(* Logix 5000 project; controller p65 vendor 1 type 14 code 85 rev 20.11; software revision 20.01; part 5 of 7 *)
(* tags used below, declared in another part *)
   DCMicroGridisInOperation : ALIAS FOR DINT00_23.8;
   DCMicroGridisSimulating : ALIAS FOR DINT00_23.10;
   House05accountBalance : ALIAS FOR REAL00_167;
   House05accountDepositRate : ALIAS FOR REAL00_168;
   House05Bclose : ALIAS FOR Local:3:O.Data.4;
   House05BcloseHILS : ALIAS FOR plc1_local_6[0].4;
   House05BcloseProxy : ALIAS FOR DINT00_31.1;
   House05BintReqClose : ALIAS FOR DINT00_31.2;
   House05BisClosed : ALIAS FOR DINT00_31.3;
   House05BisOpen : ALIAS FOR DINT00_31.4;
   House05BreqClose : ALIAS FOR DINT00_31.5;
   House05BreqOpen : ALIAS FOR DINT00_31.6;
   House05commandChanged : ALIAS FOR DINT00_31.7;
   House05commandChangedTimer : ALIAS FOR CLTIMER00_78;
   House05current : ALIAS FOR REAL00_169;
   House05currentHILS : ALIAS FOR plc1_local_2[4];
   House05currentRaw : ALIAS FOR Local:2:I.Ch0Data;
   House05deadband : ALIAS FOR REAL00_170;
   House05depositTimer : ALIAS FOR CLTIMER00_79;
   House05DisconnectPowerEventFail : ALIAS FOR DINT00_31.8;
   House05DisconnectPowerEventSuccess : ALIAS FOR DINT00_31.9;
   House05DisconnectPowerFailTimer : ALIAS FOR CLTIMER00_80;
   House05DisconnectPowerInProcess : ALIAS FOR DINT00_31.10;
   House05DisconnectPowerMsg : ALIAS FOR MESSAGE00_20;
   House05DisconnectPowerSuccessTimer : ALIAS FOR CLTIMER00_81;
   House05failedToConnect : ALIAS FOR DINT00_31.11;
   House05failedToDisconnect : ALIAS FOR DINT00_31.12;
   House05fundsAvailable : ALIAS FOR DINT00_31.13;
   House05incrementToAdd : ALIAS FOR REAL00_171;
   House05incrementToSubtract : ALIAS FOR REAL00_172;
   House05intReqConnect : ALIAS FOR DINT00_31.14;
   House05isConnected : ALIAS FOR DINT00_31.15;
   House05isDisconnected : ALIAS FOR DINT00_31.16;
   House05minBalance : ALIAS FOR REAL00_174;
   House05minBalanceToReconnect : ALIAS FOR REAL00_175;
   House05minTime : ALIAS FOR REAL00_176;
   House05powerRate : ALIAS FOR REAL00_177;
   House05powerRateMax : REAL;
   House05PurchasePowerEventFail : ALIAS FOR DINT00_31.17;
   House05PurchasePowerEventSuccess : ALIAS FOR DINT00_31.18;
   House05PurchasePowerFailTimer : ALIAS FOR CLTIMER00_82;
   House05PurchasePowerInProcess : ALIAS FOR DINT00_31.19;
   House05PurchasePowerMsg : ALIAS FOR MESSAGE00_21;
   House05PurchasePowerSuccessTimer : ALIAS FOR CLTIMER00_83;
   House05reqConnect : ALIAS FOR DINT00_31.20;
   House05reqDisconnect : ALIAS FOR DINT00_31.21;
   House05runningOut : ALIAS FOR DINT00_31.22;
   House05spendingRate : ALIAS FOR REAL00_178;
   House05timeRemaining : ALIAS FOR REAL00_179;
   House05usageTimer : ALIAS FOR CLTIMER00_84;
   Load01accountBalance : ALIAS FOR REAL00_37;
   Load01accountDepositRate : ALIAS FOR REAL00_38;
   Load01Bclose : ALIAS FOR Local:3:O.Data.5;
   Load01BcloseHILS : ALIAS FOR plc1_local_6[0].5;
   Load01BcloseProxy : ALIAS FOR DINT00_23.31;
   Load01BintReqClose : ALIAS FOR DINT00_24.0;
   Load01BisClosed : ALIAS FOR DINT00_24.1;
   Load01BisOpen : ALIAS FOR DINT00_24.2;
   Load01BreqClose : ALIAS FOR DINT00_24.3;
   Load01BreqOpen : ALIAS FOR DINT00_24.4;
   Load01commandChanged : ALIAS FOR DINT00_24.5;
   Load01commandChangedTimer : ALIAS FOR CLTIMER00_9;
   Load01current : ALIAS FOR REAL00_39;
   Load01currentHILS : ALIAS FOR plc1_local_2[5];
   Load01currentRaw : ALIAS FOR Local:2:I.Ch2Data;
   Load01deadband : ALIAS FOR REAL00_40;
   Load01depositTimer : ALIAS FOR CLTIMER00_10;
   Load01DisconnectPowerEventFail : ALIAS FOR DINT00_24.6;
   Load01DisconnectPowerEventSuccess : ALIAS FOR DINT00_24.7;
   Load01DisconnectPowerFailTimer : ALIAS FOR CLTIMER00_11;
   Load01DisconnectPowerInProcess : ALIAS FOR DINT00_24.8;
   Load01DisconnectPowerMsg : ALIAS FOR MESSAGE00_1;
   Load01DisconnectPowerSuccessTimer : ALIAS FOR CLTIMER00_12;
   Load01failedToConnect : ALIAS FOR DINT00_24.9;
   Load01failedToDisconnect : ALIAS FOR DINT00_24.10;
   Load01fundsAvailable : ALIAS FOR DINT00_24.11;
   Load01incrementToAdd : ALIAS FOR REAL00_41;
   Load01incrementToSubtract : ALIAS FOR REAL00_42;
   Load01intReqConnect : ALIAS FOR DINT00_24.12;
   Load01isConnected : ALIAS FOR DINT00_24.13;
   Load01isDisconnected : ALIAS FOR DINT00_24.14;
   Load01minBalance : ALIAS FOR REAL00_44;
   Load01minBalanceToReconnect : ALIAS FOR REAL00_45;
   Load01minTime : ALIAS FOR REAL00_46;
   Load01powerRate : ALIAS FOR REAL00_47;
   Load01powerRateMax : REAL;
   Load01PurchasePowerEventFail : ALIAS FOR DINT00_24.15;
   Load01PurchasePowerEventSuccess : ALIAS FOR DINT00_24.16;
   Load01PurchasePowerFailTimer : ALIAS FOR CLTIMER00_13;
   Load01PurchasePowerInProcess : ALIAS FOR DINT00_24.17;
   Load01PurchasePowerMsg : ALIAS FOR MESSAGE00_2;
   Load01PurchasePowerSuccessTimer : ALIAS FOR CLTIMER00_14;
   Load01reqConnect : ALIAS FOR DINT00_24.18;
   Load01reqDisconnect : ALIAS FOR DINT00_24.19;
   Load01runningOut : ALIAS FOR DINT00_24.20;
   Load01spendingRate : ALIAS FOR REAL00_48;
   Load01timeRemaining : ALIAS FOR REAL00_49;
   Load01usageTimer : ALIAS FOR CLTIMER00_15;
   Load02accountBalance : ALIAS FOR REAL00_50;
   Load02accountDepositRate : ALIAS FOR REAL00_51;
   Load02Bclose : ALIAS FOR Local:3:O.Data.6;
   Load02BcloseHILS : ALIAS FOR plc1_local_6[0].6;
   Load02BcloseProxy : ALIAS FOR DINT00_24.21;
   Load02BintReqClose : ALIAS FOR DINT00_24.22;
   Load02BisClosed : ALIAS FOR DINT00_24.23;
   Load02BisOpen : ALIAS FOR DINT00_24.24;
   Load02BreqClose : ALIAS FOR DINT00_24.25;
   Load02BreqOpen : ALIAS FOR DINT00_24.26;
   Load02commandChanged : ALIAS FOR DINT00_24.27;
   Load02commandChangedTimer : ALIAS FOR CLTIMER00_16;
   Load02current : ALIAS FOR REAL00_52;
   Load02currentHILS : ALIAS FOR plc1_local_2[6];
   Load02currentRaw : ALIAS FOR Local:2:I.Ch3Data;
   Load02deadband : ALIAS FOR REAL00_53;
   Load02depositTimer : ALIAS FOR CLTIMER00_17;
   Load02DisconnectPowerEventFail : ALIAS FOR DINT00_24.28;
   Load02DisconnectPowerEventSuccess : ALIAS FOR DINT00_24.29;
   Load02DisconnectPowerFailTimer : ALIAS FOR CLTIMER00_18;
   Load02DisconnectPowerInProcess : ALIAS FOR DINT00_24.30;
   Load02DisconnectPowerMsg : ALIAS FOR MESSAGE00_3;
   Load02DisconnectPowerSuccessTimer : ALIAS FOR CLTIMER00_19;
   Load02failedToConnect : ALIAS FOR DINT00_24.31;
   Load02failedToDisconnect : ALIAS FOR DINT00_25.0;
   Load02fundsAvailable : ALIAS FOR DINT00_25.1;
   Load02incrementToAdd : ALIAS FOR REAL00_54;
   Load02incrementToSubtract : ALIAS FOR REAL00_55;
   Load02intReqConnect : ALIAS FOR DINT00_25.2;
   Load02isConnected : ALIAS FOR DINT00_25.3;
   Load02isDisconnected : ALIAS FOR DINT00_25.4;
   Load02minBalance : ALIAS FOR REAL00_57;
   Load02minBalanceToReconnect : ALIAS FOR REAL00_58;
   Load02minTime : ALIAS FOR REAL00_59;
   Load02powerRate : ALIAS FOR REAL00_60;
   Load02powerRateMax : REAL;
   Load02PurchasePowerEventFail : ALIAS FOR DINT00_25.5;
   Load02PurchasePowerEventSuccess : ALIAS FOR DINT00_25.6;
   Load02PurchasePowerFailTimer : ALIAS FOR CLTIMER00_20;
   Load02PurchasePowerInProcess : ALIAS FOR DINT00_25.7;
   Load02PurchasePowerMsg : ALIAS FOR MESSAGE00_4;
   Load02PurchasePowerSuccessTimer : ALIAS FOR CLTIMER00_21;
   Load02reqConnect : ALIAS FOR DINT00_25.8;
   Load02reqDisconnect : ALIAS FOR DINT00_25.9;
   Load02runningOut : ALIAS FOR DINT00_25.10;
   Load02spendingRate : ALIAS FOR REAL00_61;
   Load02timeRemaining : ALIAS FOR REAL00_62;
   Load02usageTimer : ALIAS FOR CLTIMER00_22;
   LoadslowVoltage : ALIAS FOR DINT00_27.23;
   UsingAgents : BOOL;

PROGRAM House05   (* main routine House05 *)

ROUTINE House05   (* ladder *)
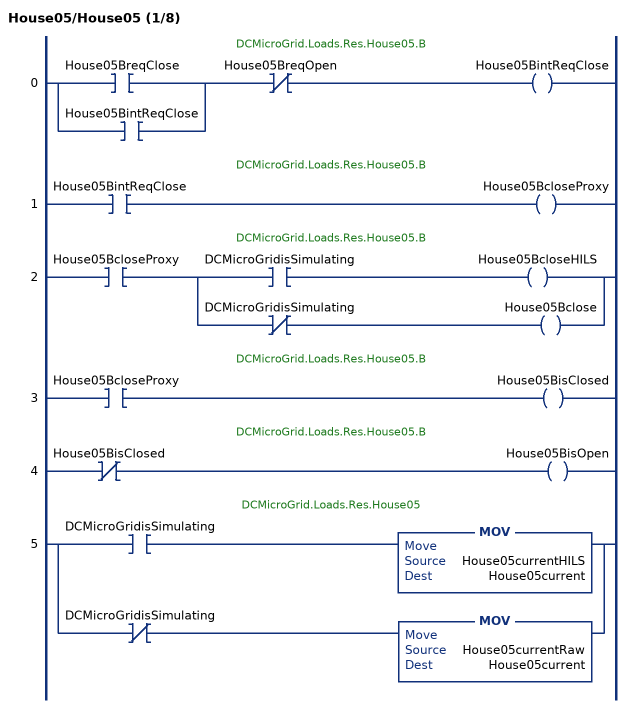
   // DCMicroGrid.Loads.Res.House05.B
   0: [XIC(House05BreqClose) ,XIC(House05BintReqClose) ]XIO(House05BreqOpen)OTE(House05BintReqClose);
   // DCMicroGrid.Loads.Res.House05.B
   1: XIC(House05BintReqClose)OTE(House05BcloseProxy);
   // DCMicroGrid.Loads.Res.House05.B
   2: XIC(House05BcloseProxy)[XIC(DCMicroGridisSimulating) OTE(House05BcloseHILS) ,XIO(DCMicroGridisSimulating) OTE(House05Bclose) ];
   // DCMicroGrid.Loads.Res.House05.B
   3: XIC(House05BcloseProxy)OTE(House05BisClosed);
   // DCMicroGrid.Loads.Res.House05.B
   4: XIO(House05BisClosed)OTE(House05BisOpen);
   // DCMicroGrid.Loads.Res.House05
   5: [XIC(DCMicroGridisSimulating) MOV(House05currentHILS,House05current) ,XIO(DCMicroGridisSimulating) MOV(House05currentRaw,House05current) ];
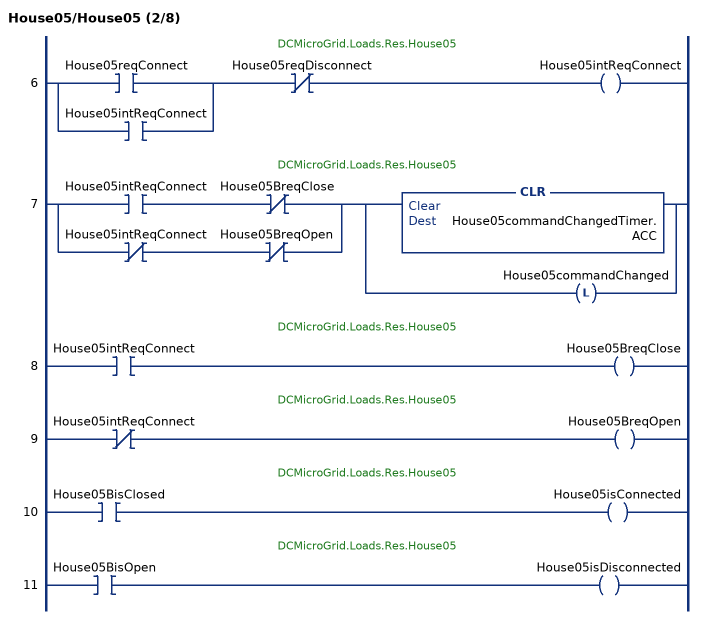
   // DCMicroGrid.Loads.Res.House05
   6: [XIC(House05reqConnect) ,XIC(House05intReqConnect) ]XIO(House05reqDisconnect)OTE(House05intReqConnect);
   // DCMicroGrid.Loads.Res.House05
   7: [XIC(House05intReqConnect) XIO(House05BreqClose) ,XIO(House05intReqConnect) XIO(House05BreqOpen) ][CLR(House05commandChangedTimer.ACC) ,OTL(House05commandChanged) ];
   // DCMicroGrid.Loads.Res.House05
   8: XIC(House05intReqConnect)OTE(House05BreqClose);
   // DCMicroGrid.Loads.Res.House05
   9: XIO(House05intReqConnect)OTE(House05BreqOpen);
   // DCMicroGrid.Loads.Res.House05
   10: XIC(House05BisClosed)OTE(House05isConnected);
   // DCMicroGrid.Loads.Res.House05
   11: XIC(House05BisOpen)OTE(House05isDisconnected);
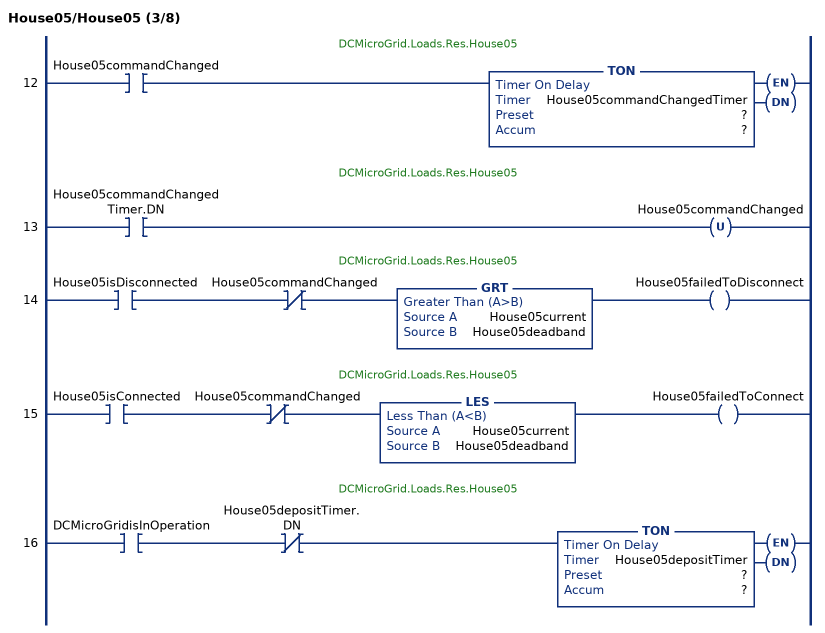
   // DCMicroGrid.Loads.Res.House05
   12: XIC(House05commandChanged)TON(House05commandChangedTimer,?,?);
   // DCMicroGrid.Loads.Res.House05
   13: XIC(House05commandChangedTimer.DN)OTU(House05commandChanged);
   // DCMicroGrid.Loads.Res.House05
   14: XIC(House05isDisconnected)XIO(House05commandChanged)GRT(House05current,House05deadband)OTE(House05failedToDisconnect);
   // DCMicroGrid.Loads.Res.House05
   15: XIC(House05isConnected)XIO(House05commandChanged)LES(House05current,House05deadband)OTE(House05failedToConnect);
   // DCMicroGrid.Loads.Res.House05
   16: XIC(DCMicroGridisInOperation)XIO(House05depositTimer.DN)TON(House05depositTimer,?,?);
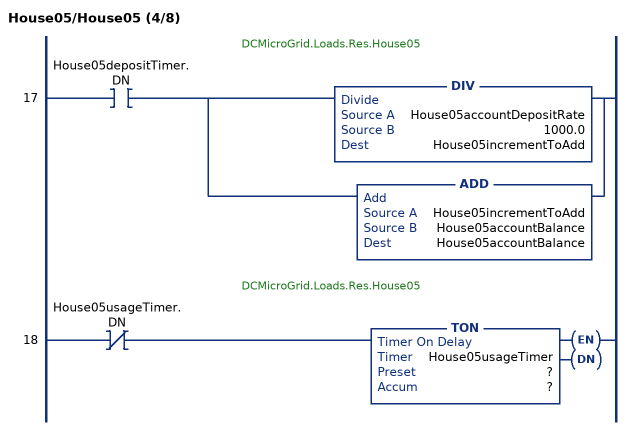
   // DCMicroGrid.Loads.Res.House05
   17: XIC(House05depositTimer.DN)[DIV(House05accountDepositRate,1000.0,House05incrementToAdd) ,ADD(House05incrementToAdd,House05accountBalance,House05accountBalance) ];
   // DCMicroGrid.Loads.Res.House05
   18: XIO(House05usageTimer.DN)TON(House05usageTimer,?,?);
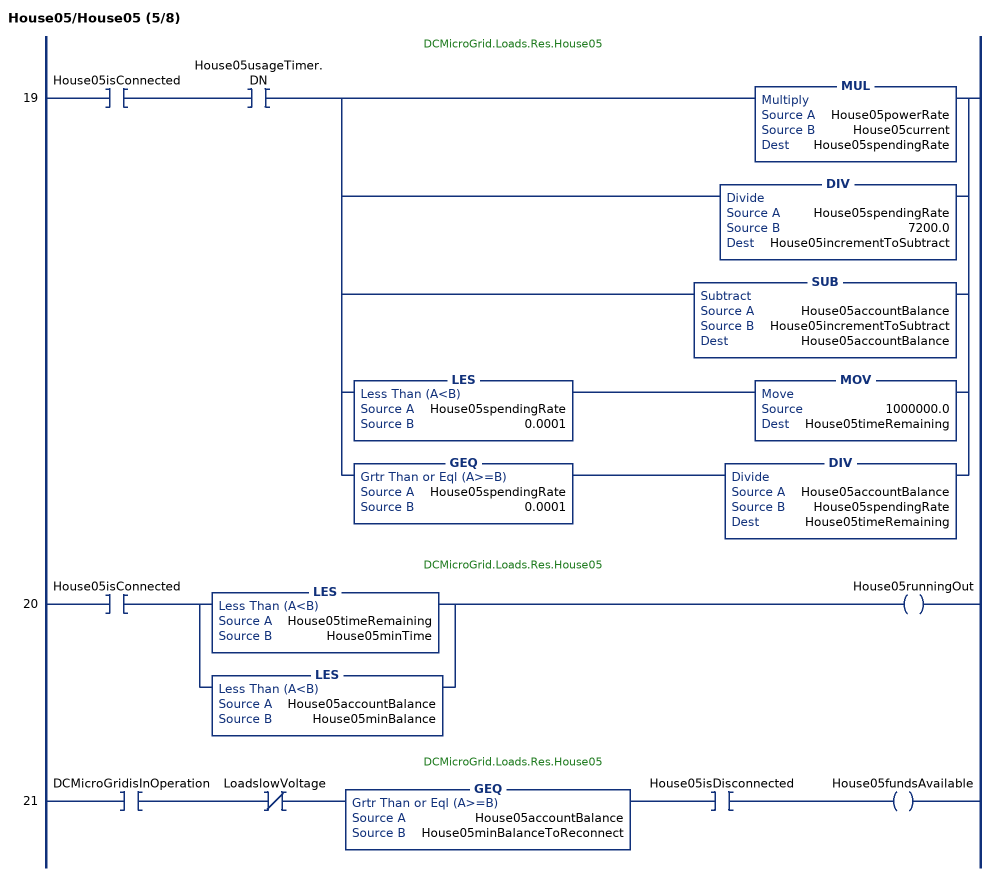
   // DCMicroGrid.Loads.Res.House05
   19: XIC(House05isConnected)XIC(House05usageTimer.DN)[MUL(House05powerRate,House05current,House05spendingRate) ,DIV(House05spendingRate,7200.0,House05incrementToSubtract) ,SUB(House05accountBalance,House05incrementToSubtract,House05accountBalance) ,[LES(House05spendingRate,0.0001) MOV(1000000.0,House05timeRemaining) ,GEQ(House05spendingRate,0.0001) DIV(House05accountBalance,House05spendingRate,House05timeRemaining) ] ];
   // DCMicroGrid.Loads.Res.House05
   20: XIC(House05isConnected)[LES(House05timeRemaining,House05minTime) ,LES(House05accountBalance,House05minBalance) ]OTE(House05runningOut);
   // DCMicroGrid.Loads.Res.House05
   21: XIC(DCMicroGridisInOperation)XIO(LoadslowVoltage)GEQ(House05accountBalance,House05minBalanceToReconnect)XIC(House05isDisconnected)OTE(House05fundsAvailable);
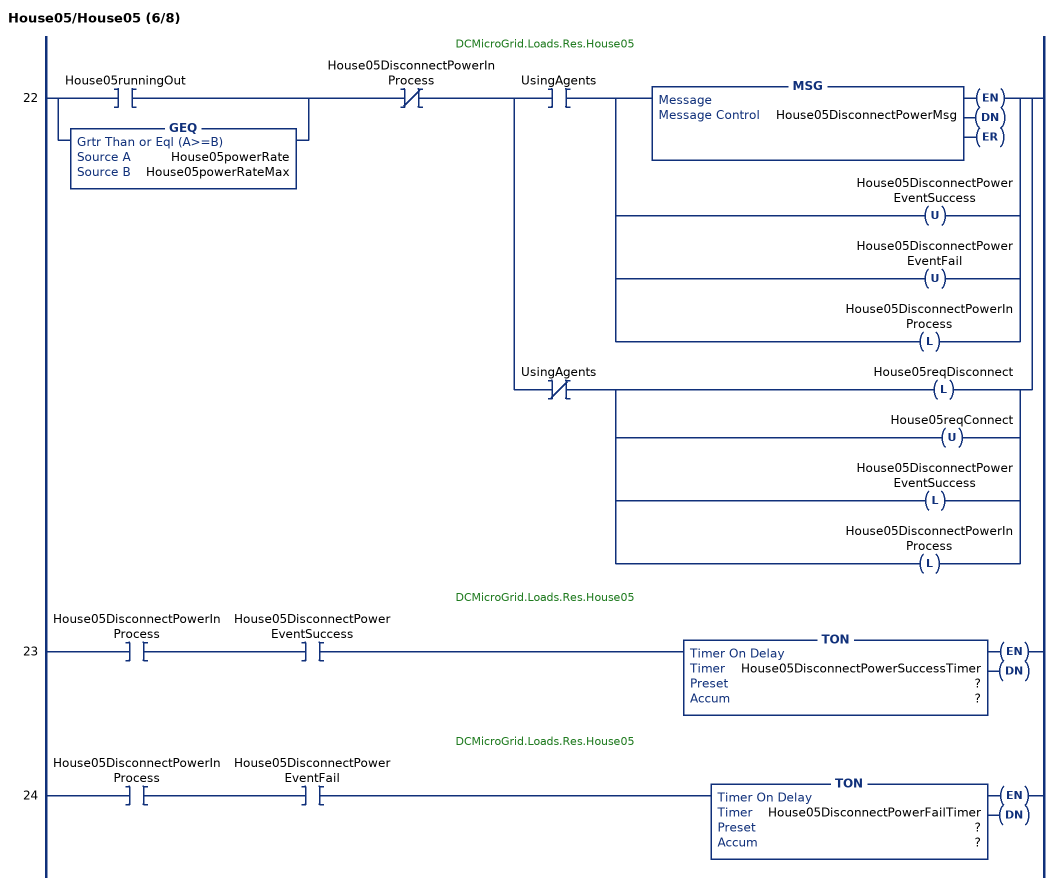
   // DCMicroGrid.Loads.Res.House05
   22: [XIC(House05runningOut) ,GEQ(House05powerRate,House05powerRateMax) ]XIO(House05DisconnectPowerInProcess)[XIC(UsingAgents) [MSG(House05DisconnectPowerMsg) ,OTU(House05DisconnectPowerEventSuccess) ,OTU(House05DisconnectPowerEventFail) ,OTL(House05DisconnectPowerInProcess) ] ,XIO(UsingAgents) [OTL(House05reqDisconnect) ,OTU(House05reqConnect) ,OTL(House05DisconnectPowerEventSuccess) ,OTL(House05DisconnectPowerInProcess) ] ];
   // DCMicroGrid.Loads.Res.House05
   23: XIC(House05DisconnectPowerInProcess)XIC(House05DisconnectPowerEventSuccess)TON(House05DisconnectPowerSuccessTimer,?,?);
   // DCMicroGrid.Loads.Res.House05
   24: XIC(House05DisconnectPowerInProcess)XIC(House05DisconnectPowerEventFail)TON(House05DisconnectPowerFailTimer,?,?);
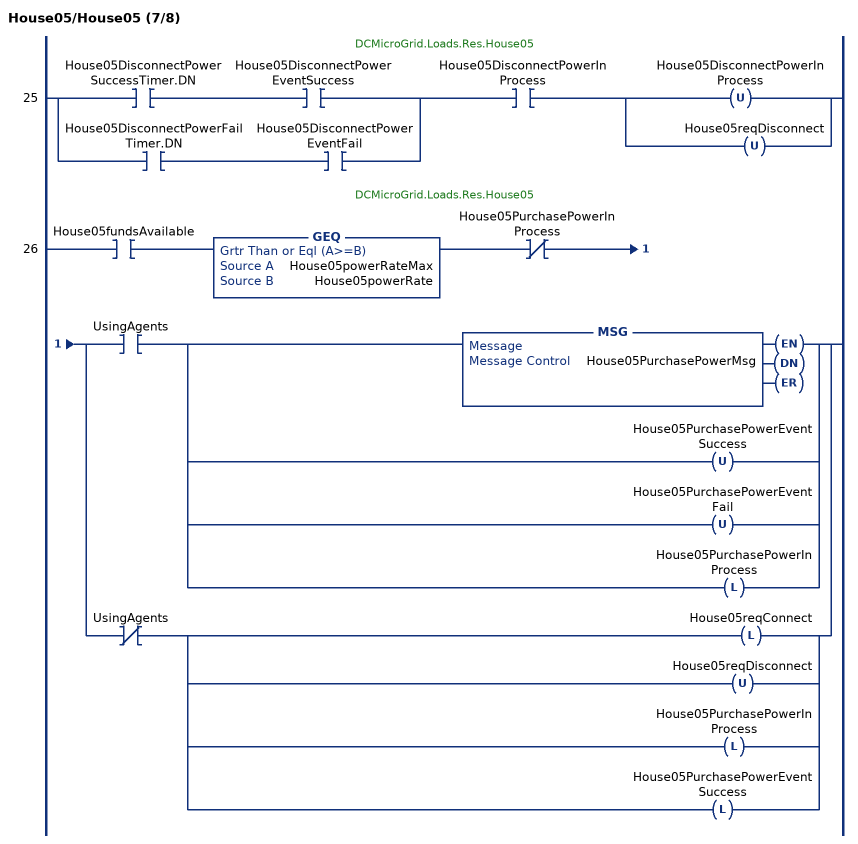
   // DCMicroGrid.Loads.Res.House05
   25: [XIC(House05DisconnectPowerSuccessTimer.DN) XIC(House05DisconnectPowerEventSuccess) ,XIC(House05DisconnectPowerFailTimer.DN) XIC(House05DisconnectPowerEventFail) ]XIC(House05DisconnectPowerInProcess)[OTU(House05DisconnectPowerInProcess) ,OTU(House05reqDisconnect) ];
   // DCMicroGrid.Loads.Res.House05
   26: XIC(House05fundsAvailable)GEQ(House05powerRateMax,House05powerRate)XIO(House05PurchasePowerInProcess)[XIC(UsingAgents) [MSG(House05PurchasePowerMsg) ,OTU(House05PurchasePowerEventSuccess) ,OTU(House05PurchasePowerEventFail) ,OTL(House05PurchasePowerInProcess) ] ,XIO(UsingAgents) [OTL(House05reqConnect) ,OTU(House05reqDisconnect) ,OTL(House05PurchasePowerInProcess) ,OTL(House05PurchasePowerEventSuccess) ] ];
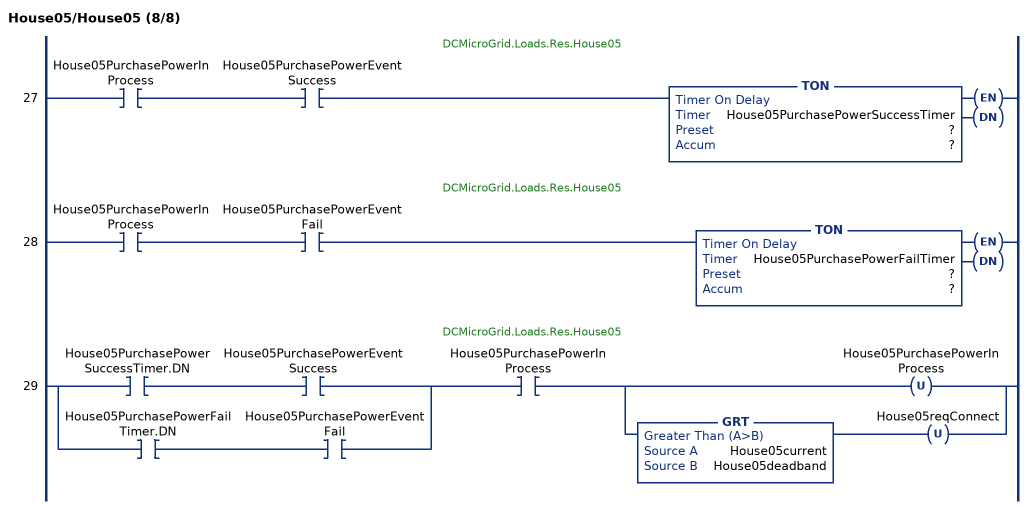
   // DCMicroGrid.Loads.Res.House05
   27: XIC(House05PurchasePowerInProcess)XIC(House05PurchasePowerEventSuccess)TON(House05PurchasePowerSuccessTimer,?,?);
   // DCMicroGrid.Loads.Res.House05
   28: XIC(House05PurchasePowerInProcess)XIC(House05PurchasePowerEventFail)TON(House05PurchasePowerFailTimer,?,?);
   // DCMicroGrid.Loads.Res.House05
   29: [XIC(House05PurchasePowerSuccessTimer.DN) XIC(House05PurchasePowerEventSuccess) ,XIC(House05PurchasePowerFailTimer.DN) XIC(House05PurchasePowerEventFail) ]XIC(House05PurchasePowerInProcess)[OTU(House05PurchasePowerInProcess) ,GRT(House05current,House05deadband) OTU(House05reqConnect) ];
END_ROUTINE
END_PROGRAM

PROGRAM Load01   (* main routine Load01 *)

ROUTINE Load01   (* ladder *)
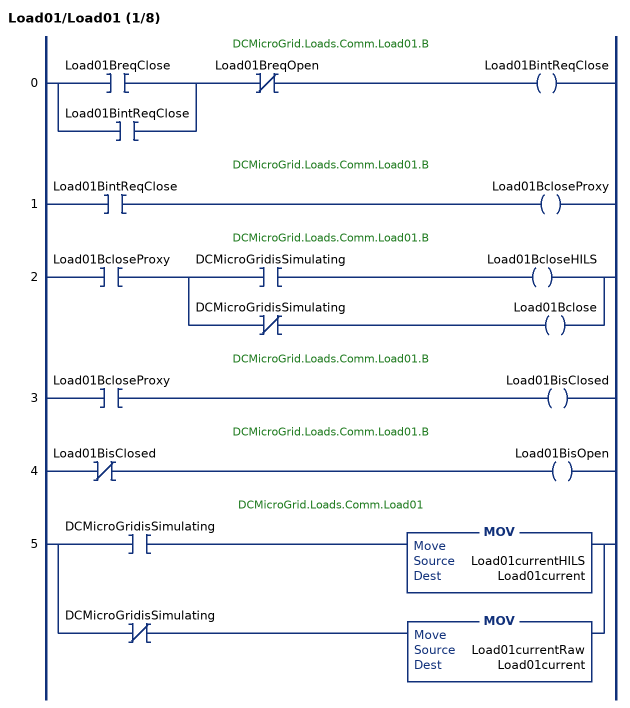
   // DCMicroGrid.Loads.Comm.Load01.B
   0: [XIC(Load01BreqClose) ,XIC(Load01BintReqClose) ]XIO(Load01BreqOpen)OTE(Load01BintReqClose);
   // DCMicroGrid.Loads.Comm.Load01.B
   1: XIC(Load01BintReqClose)OTE(Load01BcloseProxy);
   // DCMicroGrid.Loads.Comm.Load01.B
   2: XIC(Load01BcloseProxy)[XIC(DCMicroGridisSimulating) OTE(Load01BcloseHILS) ,XIO(DCMicroGridisSimulating) OTE(Load01Bclose) ];
   // DCMicroGrid.Loads.Comm.Load01.B
   3: XIC(Load01BcloseProxy)OTE(Load01BisClosed);
   // DCMicroGrid.Loads.Comm.Load01.B
   4: XIO(Load01BisClosed)OTE(Load01BisOpen);
   // DCMicroGrid.Loads.Comm.Load01
   5: [XIC(DCMicroGridisSimulating) MOV(Load01currentHILS,Load01current) ,XIO(DCMicroGridisSimulating) MOV(Load01currentRaw,Load01current) ];
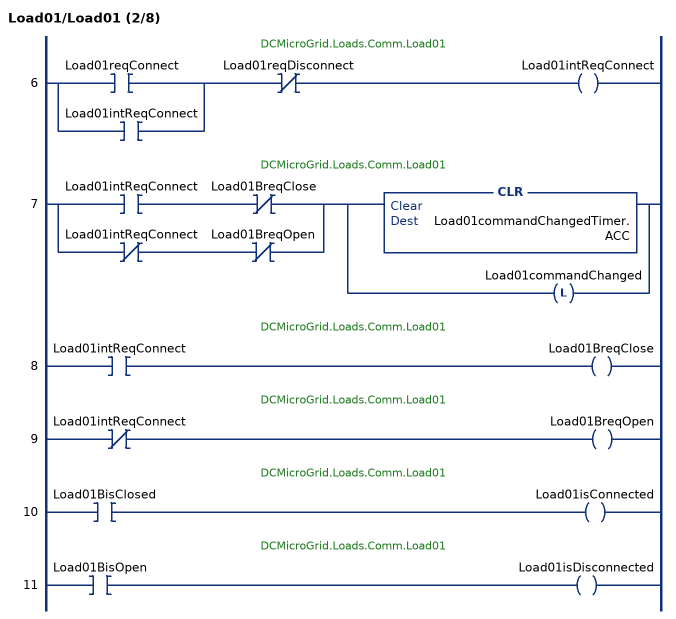
   // DCMicroGrid.Loads.Comm.Load01
   6: [XIC(Load01reqConnect) ,XIC(Load01intReqConnect) ]XIO(Load01reqDisconnect)OTE(Load01intReqConnect);
   // DCMicroGrid.Loads.Comm.Load01
   7: [XIC(Load01intReqConnect) XIO(Load01BreqClose) ,XIO(Load01intReqConnect) XIO(Load01BreqOpen) ][CLR(Load01commandChangedTimer.ACC) ,OTL(Load01commandChanged) ];
   // DCMicroGrid.Loads.Comm.Load01
   8: XIC(Load01intReqConnect)OTE(Load01BreqClose);
   // DCMicroGrid.Loads.Comm.Load01
   9: XIO(Load01intReqConnect)OTE(Load01BreqOpen);
   // DCMicroGrid.Loads.Comm.Load01
   10: XIC(Load01BisClosed)OTE(Load01isConnected);
   // DCMicroGrid.Loads.Comm.Load01
   11: XIC(Load01BisOpen)OTE(Load01isDisconnected);
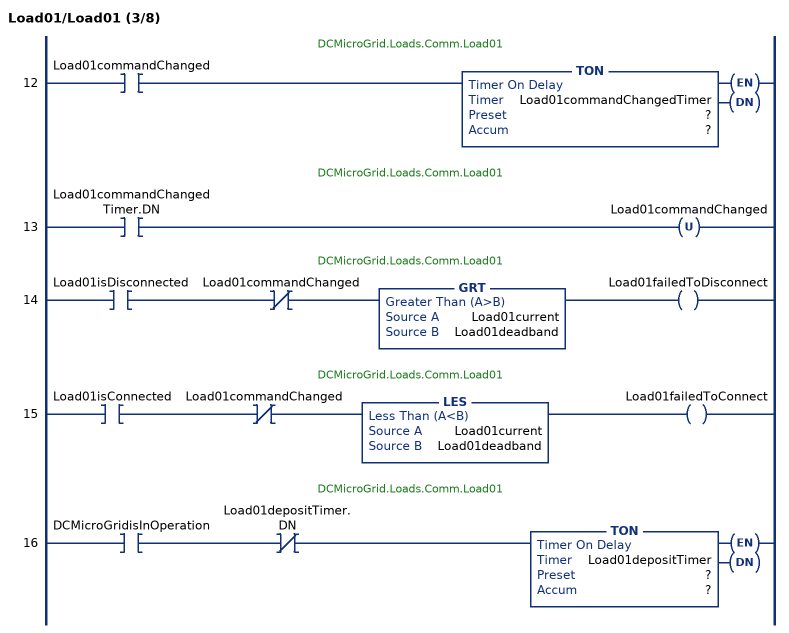
   // DCMicroGrid.Loads.Comm.Load01
   12: XIC(Load01commandChanged)TON(Load01commandChangedTimer,?,?);
   // DCMicroGrid.Loads.Comm.Load01
   13: XIC(Load01commandChangedTimer.DN)OTU(Load01commandChanged);
   // DCMicroGrid.Loads.Comm.Load01
   14: XIC(Load01isDisconnected)XIO(Load01commandChanged)GRT(Load01current,Load01deadband)OTE(Load01failedToDisconnect);
   // DCMicroGrid.Loads.Comm.Load01
   15: XIC(Load01isConnected)XIO(Load01commandChanged)LES(Load01current,Load01deadband)OTE(Load01failedToConnect);
   // DCMicroGrid.Loads.Comm.Load01
   16: XIC(DCMicroGridisInOperation)XIO(Load01depositTimer.DN)TON(Load01depositTimer,?,?);
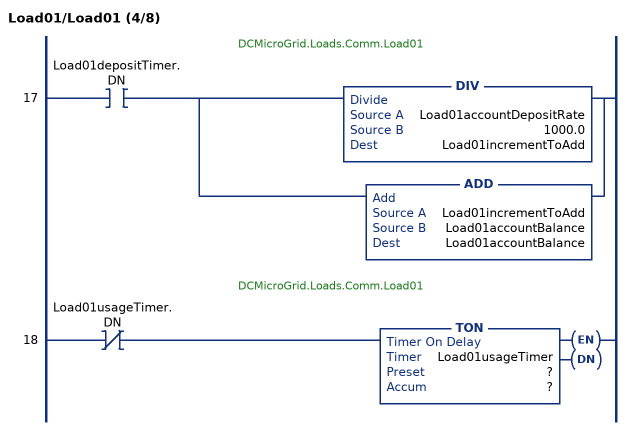
   // DCMicroGrid.Loads.Comm.Load01
   17: XIC(Load01depositTimer.DN)[DIV(Load01accountDepositRate,1000.0,Load01incrementToAdd) ,ADD(Load01incrementToAdd,Load01accountBalance,Load01accountBalance) ];
   // DCMicroGrid.Loads.Comm.Load01
   18: XIO(Load01usageTimer.DN)TON(Load01usageTimer,?,?);
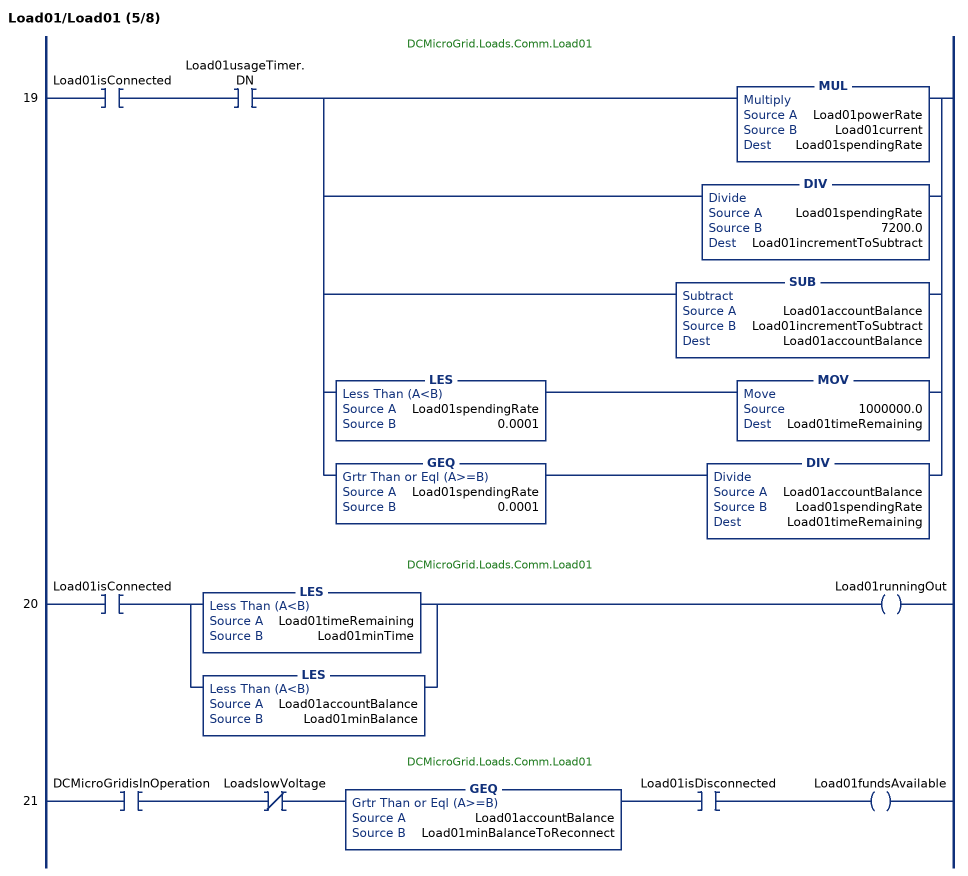
   // DCMicroGrid.Loads.Comm.Load01
   19: XIC(Load01isConnected)XIC(Load01usageTimer.DN)[MUL(Load01powerRate,Load01current,Load01spendingRate) ,DIV(Load01spendingRate,7200.0,Load01incrementToSubtract) ,SUB(Load01accountBalance,Load01incrementToSubtract,Load01accountBalance) ,[LES(Load01spendingRate,0.0001) MOV(1000000.0,Load01timeRemaining) ,GEQ(Load01spendingRate,0.0001) DIV(Load01accountBalance,Load01spendingRate,Load01timeRemaining) ] ];
   // DCMicroGrid.Loads.Comm.Load01
   20: XIC(Load01isConnected)[LES(Load01timeRemaining,Load01minTime) ,LES(Load01accountBalance,Load01minBalance) ]OTE(Load01runningOut);
   // DCMicroGrid.Loads.Comm.Load01
   21: XIC(DCMicroGridisInOperation)XIO(LoadslowVoltage)GEQ(Load01accountBalance,Load01minBalanceToReconnect)XIC(Load01isDisconnected)OTE(Load01fundsAvailable);
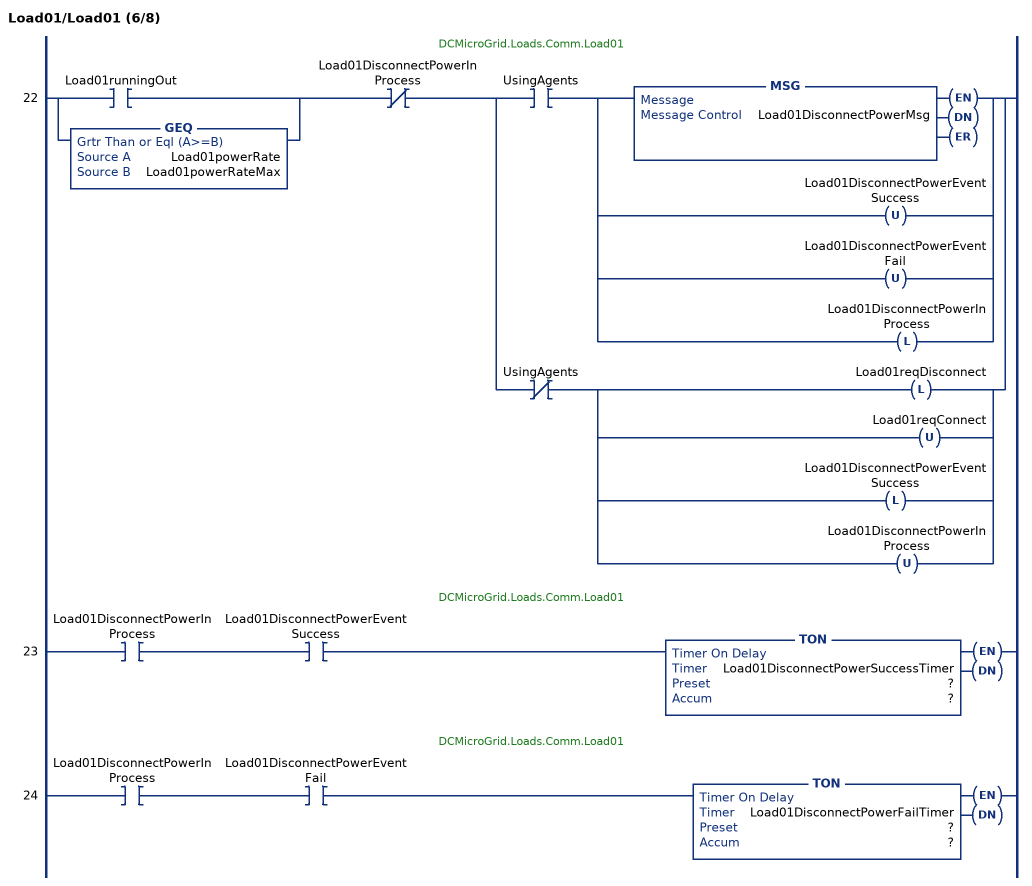
   // DCMicroGrid.Loads.Comm.Load01
   22: [XIC(Load01runningOut) ,GEQ(Load01powerRate,Load01powerRateMax) ]XIO(Load01DisconnectPowerInProcess)[XIC(UsingAgents) [MSG(Load01DisconnectPowerMsg) ,OTU(Load01DisconnectPowerEventSuccess) ,OTU(Load01DisconnectPowerEventFail) ,OTL(Load01DisconnectPowerInProcess) ] ,XIO(UsingAgents) [OTL(Load01reqDisconnect) ,OTU(Load01reqConnect) ,OTL(Load01DisconnectPowerEventSuccess) ,OTU(Load01DisconnectPowerInProcess) ] ];
   // DCMicroGrid.Loads.Comm.Load01
   23: XIC(Load01DisconnectPowerInProcess)XIC(Load01DisconnectPowerEventSuccess)TON(Load01DisconnectPowerSuccessTimer,?,?);
   // DCMicroGrid.Loads.Comm.Load01
   24: XIC(Load01DisconnectPowerInProcess)XIC(Load01DisconnectPowerEventFail)TON(Load01DisconnectPowerFailTimer,?,?);
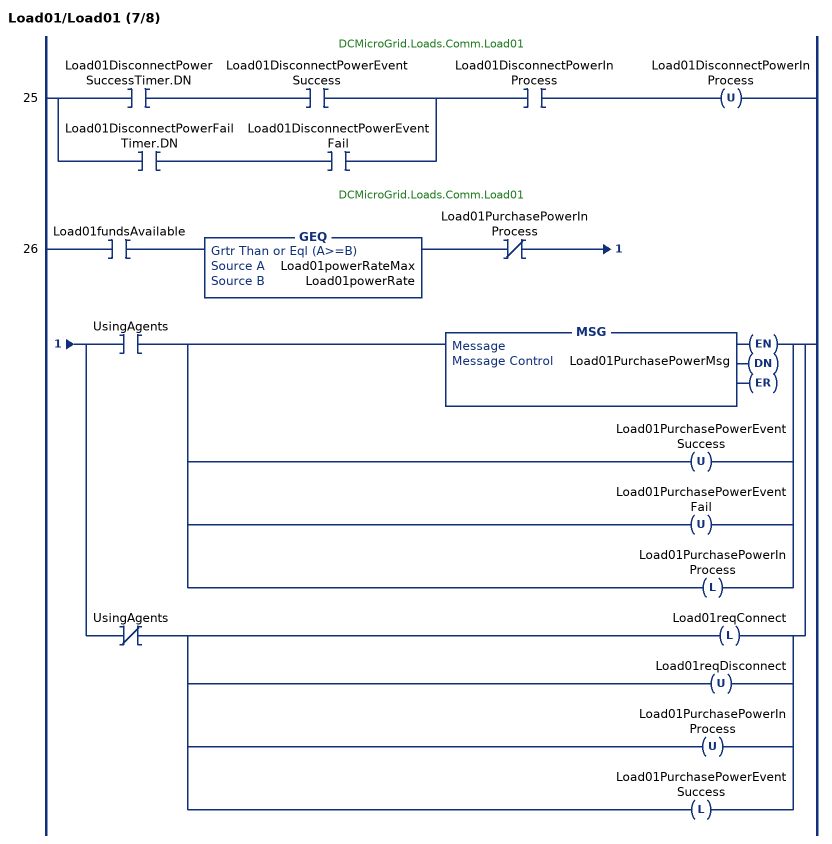
   // DCMicroGrid.Loads.Comm.Load01
   25: [XIC(Load01DisconnectPowerSuccessTimer.DN) XIC(Load01DisconnectPowerEventSuccess) ,XIC(Load01DisconnectPowerFailTimer.DN) XIC(Load01DisconnectPowerEventFail) ]XIC(Load01DisconnectPowerInProcess)OTU(Load01DisconnectPowerInProcess);
   // DCMicroGrid.Loads.Comm.Load01
   26: XIC(Load01fundsAvailable)GEQ(Load01powerRateMax,Load01powerRate)XIO(Load01PurchasePowerInProcess)[XIC(UsingAgents) [MSG(Load01PurchasePowerMsg) ,OTU(Load01PurchasePowerEventSuccess) ,OTU(Load01PurchasePowerEventFail) ,OTL(Load01PurchasePowerInProcess) ] ,XIO(UsingAgents) [OTL(Load01reqConnect) ,OTU(Load01reqDisconnect) ,OTU(Load01PurchasePowerInProcess) ,OTL(Load01PurchasePowerEventSuccess) ] ];
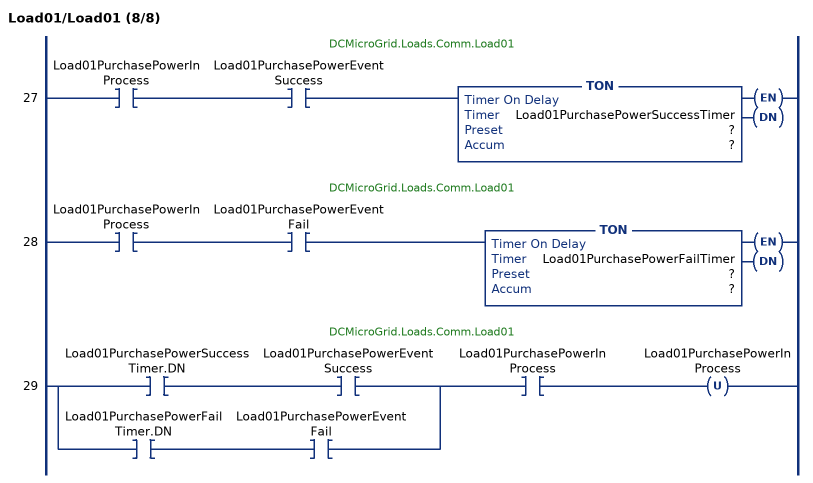
   // DCMicroGrid.Loads.Comm.Load01
   27: XIC(Load01PurchasePowerInProcess)XIC(Load01PurchasePowerEventSuccess)TON(Load01PurchasePowerSuccessTimer,?,?);
   // DCMicroGrid.Loads.Comm.Load01
   28: XIC(Load01PurchasePowerInProcess)XIC(Load01PurchasePowerEventFail)TON(Load01PurchasePowerFailTimer,?,?);
   // DCMicroGrid.Loads.Comm.Load01
   29: [XIC(Load01PurchasePowerSuccessTimer.DN) XIC(Load01PurchasePowerEventSuccess) ,XIC(Load01PurchasePowerFailTimer.DN) XIC(Load01PurchasePowerEventFail) ]XIC(Load01PurchasePowerInProcess)OTU(Load01PurchasePowerInProcess);
END_ROUTINE
END_PROGRAM

PROGRAM Load02   (* main routine Load02 *)

ROUTINE Load02   (* ladder *)
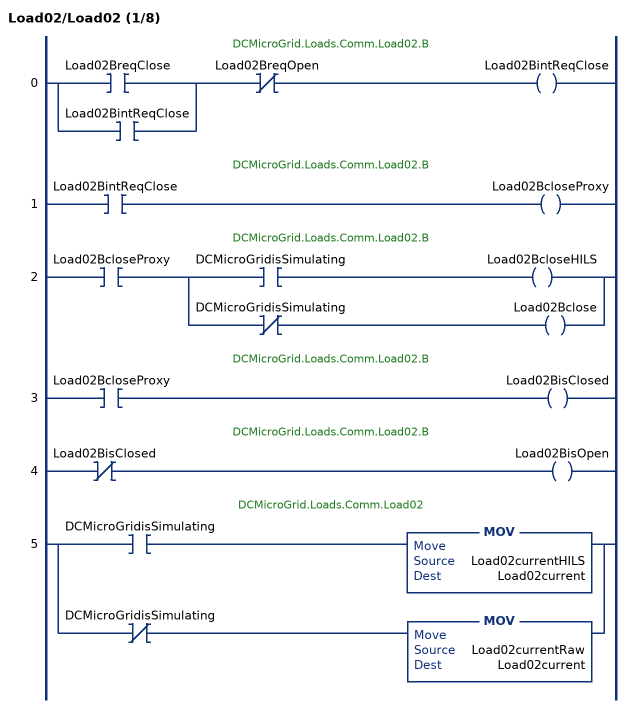
   // DCMicroGrid.Loads.Comm.Load02.B
   0: [XIC(Load02BreqClose) ,XIC(Load02BintReqClose) ]XIO(Load02BreqOpen)OTE(Load02BintReqClose);
   // DCMicroGrid.Loads.Comm.Load02.B
   1: XIC(Load02BintReqClose)OTE(Load02BcloseProxy);
   // DCMicroGrid.Loads.Comm.Load02.B
   2: XIC(Load02BcloseProxy)[XIC(DCMicroGridisSimulating) OTE(Load02BcloseHILS) ,XIO(DCMicroGridisSimulating) OTE(Load02Bclose) ];
   // DCMicroGrid.Loads.Comm.Load02.B
   3: XIC(Load02BcloseProxy)OTE(Load02BisClosed);
   // DCMicroGrid.Loads.Comm.Load02.B
   4: XIO(Load02BisClosed)OTE(Load02BisOpen);
   // DCMicroGrid.Loads.Comm.Load02
   5: [XIC(DCMicroGridisSimulating) MOV(Load02currentHILS,Load02current) ,XIO(DCMicroGridisSimulating) MOV(Load02currentRaw,Load02current) ];
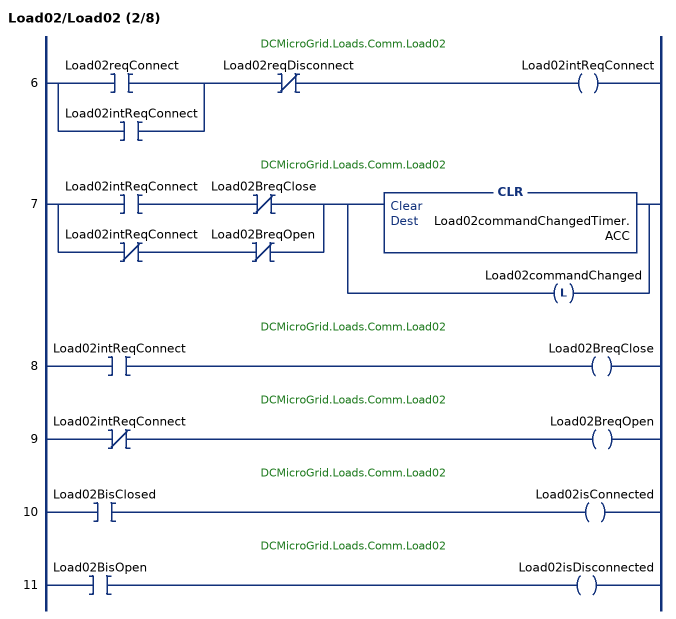
   // DCMicroGrid.Loads.Comm.Load02
   6: [XIC(Load02reqConnect) ,XIC(Load02intReqConnect) ]XIO(Load02reqDisconnect)OTE(Load02intReqConnect);
   // DCMicroGrid.Loads.Comm.Load02
   7: [XIC(Load02intReqConnect) XIO(Load02BreqClose) ,XIO(Load02intReqConnect) XIO(Load02BreqOpen) ][CLR(Load02commandChangedTimer.ACC) ,OTL(Load02commandChanged) ];
   // DCMicroGrid.Loads.Comm.Load02
   8: XIC(Load02intReqConnect)OTE(Load02BreqClose);
   // DCMicroGrid.Loads.Comm.Load02
   9: XIO(Load02intReqConnect)OTE(Load02BreqOpen);
   // DCMicroGrid.Loads.Comm.Load02
   10: XIC(Load02BisClosed)OTE(Load02isConnected);
   // DCMicroGrid.Loads.Comm.Load02
   11: XIC(Load02BisOpen)OTE(Load02isDisconnected);
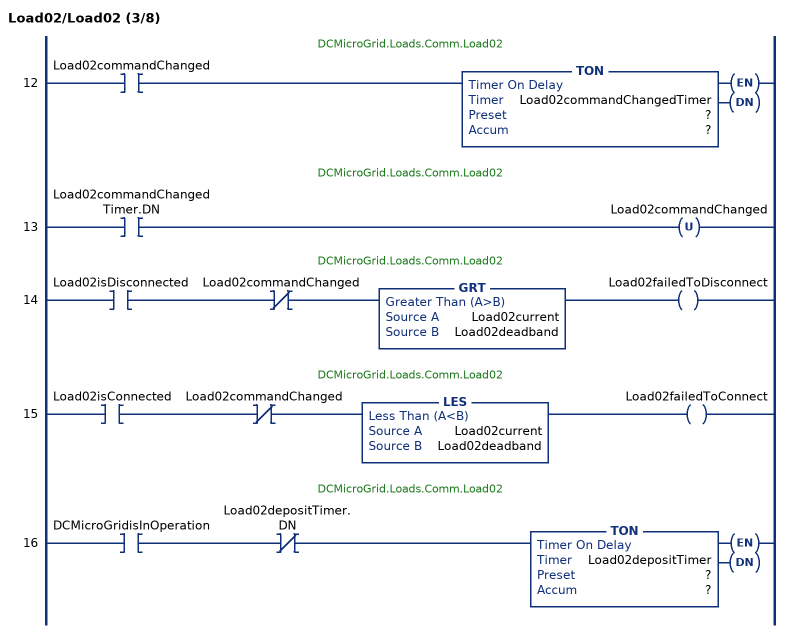
   // DCMicroGrid.Loads.Comm.Load02
   12: XIC(Load02commandChanged)TON(Load02commandChangedTimer,?,?);
   // DCMicroGrid.Loads.Comm.Load02
   13: XIC(Load02commandChangedTimer.DN)OTU(Load02commandChanged);
   // DCMicroGrid.Loads.Comm.Load02
   14: XIC(Load02isDisconnected)XIO(Load02commandChanged)GRT(Load02current,Load02deadband)OTE(Load02failedToDisconnect);
   // DCMicroGrid.Loads.Comm.Load02
   15: XIC(Load02isConnected)XIO(Load02commandChanged)LES(Load02current,Load02deadband)OTE(Load02failedToConnect);
   // DCMicroGrid.Loads.Comm.Load02
   16: XIC(DCMicroGridisInOperation)XIO(Load02depositTimer.DN)TON(Load02depositTimer,?,?);
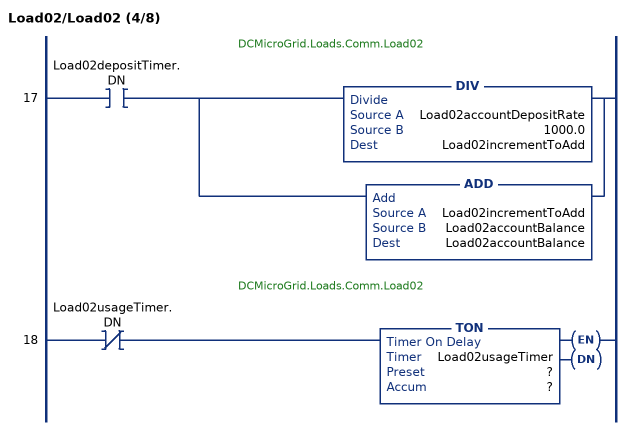
   // DCMicroGrid.Loads.Comm.Load02
   17: XIC(Load02depositTimer.DN)[DIV(Load02accountDepositRate,1000.0,Load02incrementToAdd) ,ADD(Load02incrementToAdd,Load02accountBalance,Load02accountBalance) ];
   // DCMicroGrid.Loads.Comm.Load02
   18: XIO(Load02usageTimer.DN)TON(Load02usageTimer,?,?);
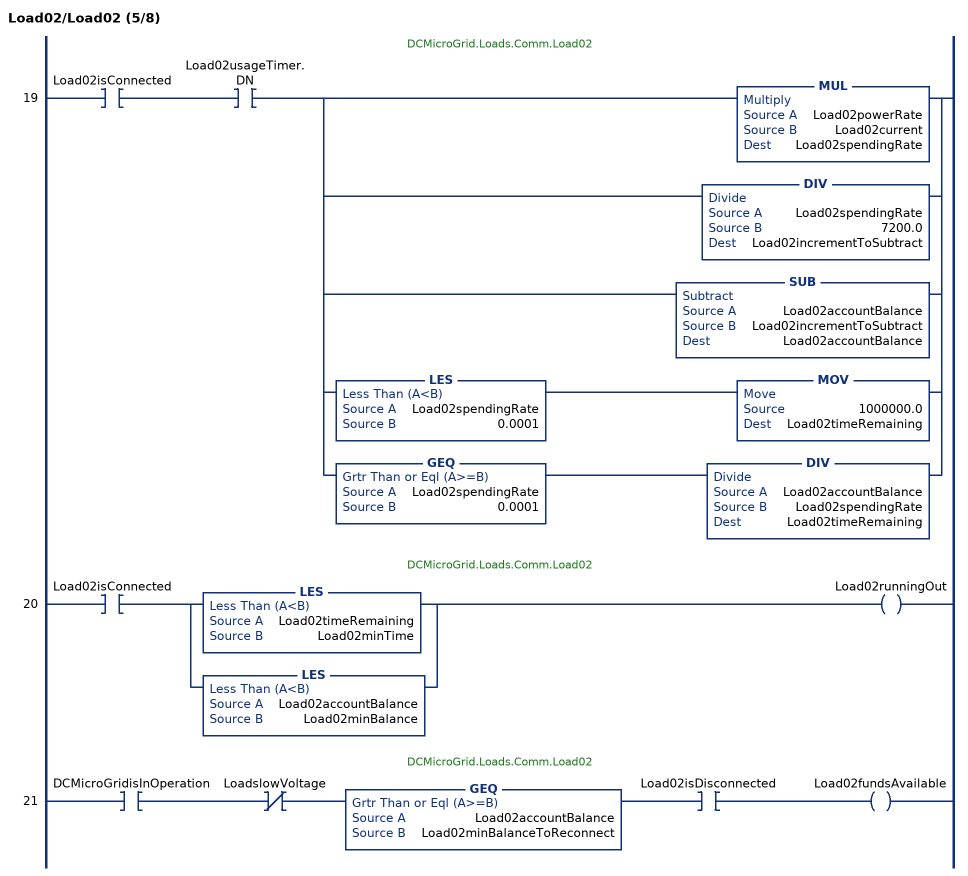
   // DCMicroGrid.Loads.Comm.Load02
   19: XIC(Load02isConnected)XIC(Load02usageTimer.DN)[MUL(Load02powerRate,Load02current,Load02spendingRate) ,DIV(Load02spendingRate,7200.0,Load02incrementToSubtract) ,SUB(Load02accountBalance,Load02incrementToSubtract,Load02accountBalance) ,[LES(Load02spendingRate,0.0001) MOV(1000000.0,Load02timeRemaining) ,GEQ(Load02spendingRate,0.0001) DIV(Load02accountBalance,Load02spendingRate,Load02timeRemaining) ] ];
   // DCMicroGrid.Loads.Comm.Load02
   20: XIC(Load02isConnected)[LES(Load02timeRemaining,Load02minTime) ,LES(Load02accountBalance,Load02minBalance) ]OTE(Load02runningOut);
   // DCMicroGrid.Loads.Comm.Load02
   21: XIC(DCMicroGridisInOperation)XIO(LoadslowVoltage)GEQ(Load02accountBalance,Load02minBalanceToReconnect)XIC(Load02isDisconnected)OTE(Load02fundsAvailable);
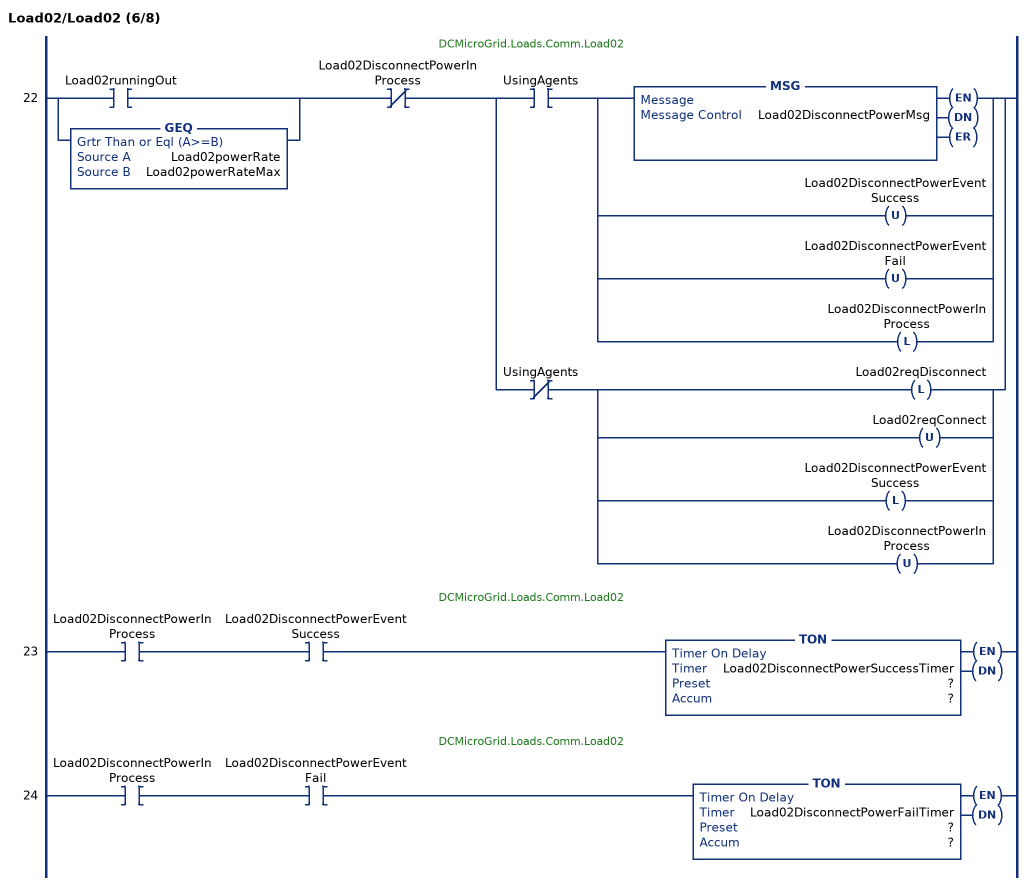
   // DCMicroGrid.Loads.Comm.Load02
   22: [XIC(Load02runningOut) ,GEQ(Load02powerRate,Load02powerRateMax) ]XIO(Load02DisconnectPowerInProcess)[XIC(UsingAgents) [MSG(Load02DisconnectPowerMsg) ,OTU(Load02DisconnectPowerEventSuccess) ,OTU(Load02DisconnectPowerEventFail) ,OTL(Load02DisconnectPowerInProcess) ] ,XIO(UsingAgents) [OTL(Load02reqDisconnect) ,OTU(Load02reqConnect) ,OTL(Load02DisconnectPowerEventSuccess) ,OTU(Load02DisconnectPowerInProcess) ] ];
   // DCMicroGrid.Loads.Comm.Load02
   23: XIC(Load02DisconnectPowerInProcess)XIC(Load02DisconnectPowerEventSuccess)TON(Load02DisconnectPowerSuccessTimer,?,?);
   // DCMicroGrid.Loads.Comm.Load02
   24: XIC(Load02DisconnectPowerInProcess)XIC(Load02DisconnectPowerEventFail)TON(Load02DisconnectPowerFailTimer,?,?);
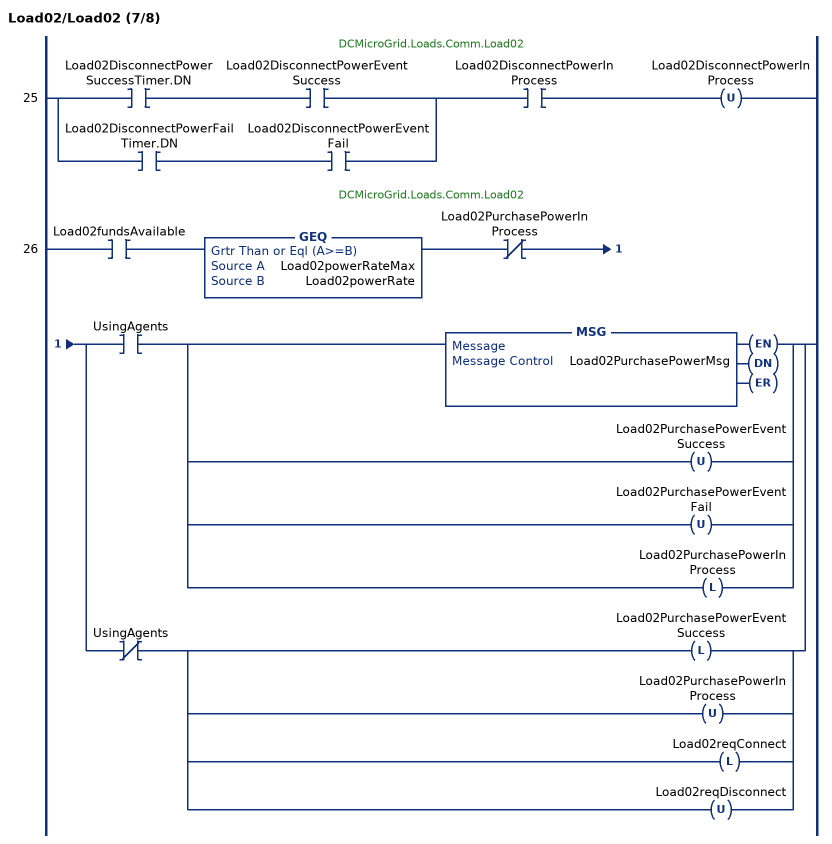
   // DCMicroGrid.Loads.Comm.Load02
   25: [XIC(Load02DisconnectPowerSuccessTimer.DN) XIC(Load02DisconnectPowerEventSuccess) ,XIC(Load02DisconnectPowerFailTimer.DN) XIC(Load02DisconnectPowerEventFail) ]XIC(Load02DisconnectPowerInProcess)OTU(Load02DisconnectPowerInProcess);
   // DCMicroGrid.Loads.Comm.Load02
   26: XIC(Load02fundsAvailable)GEQ(Load02powerRateMax,Load02powerRate)XIO(Load02PurchasePowerInProcess)[XIC(UsingAgents) [MSG(Load02PurchasePowerMsg) ,OTU(Load02PurchasePowerEventSuccess) ,OTU(Load02PurchasePowerEventFail) ,OTL(Load02PurchasePowerInProcess) ] ,XIO(UsingAgents) [OTL(Load02PurchasePowerEventSuccess) ,OTU(Load02PurchasePowerInProcess) ,OTL(Load02reqConnect) ,OTU(Load02reqDisconnect) ] ];
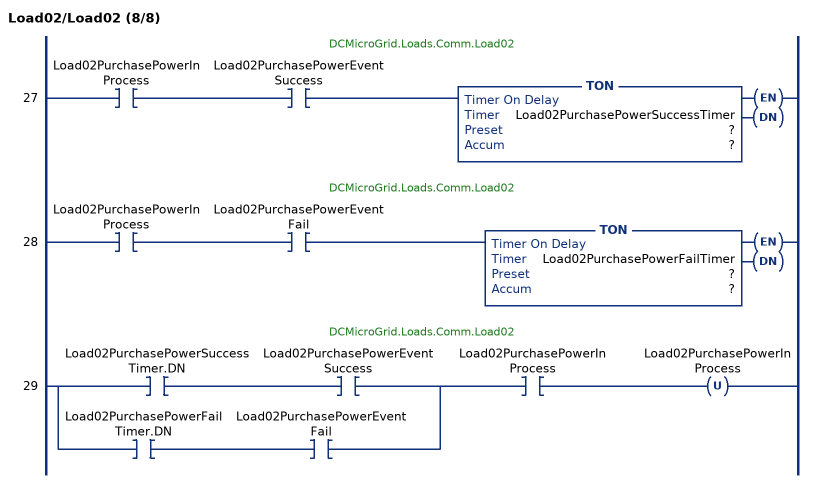
   // DCMicroGrid.Loads.Comm.Load02
   27: XIC(Load02PurchasePowerInProcess)XIC(Load02PurchasePowerEventSuccess)TON(Load02PurchasePowerSuccessTimer,?,?);
   // DCMicroGrid.Loads.Comm.Load02
   28: XIC(Load02PurchasePowerInProcess)XIC(Load02PurchasePowerEventFail)TON(Load02PurchasePowerFailTimer,?,?);
   // DCMicroGrid.Loads.Comm.Load02
   29: [XIC(Load02PurchasePowerSuccessTimer.DN) XIC(Load02PurchasePowerEventSuccess) ,XIC(Load02PurchasePowerFailTimer.DN) XIC(Load02PurchasePowerEventFail) ]XIC(Load02PurchasePowerInProcess)OTU(Load02PurchasePowerInProcess);
END_ROUTINE
END_PROGRAM
